TYPE ExampleDomain_Io_In :
STRUCT
END_STRUCT
END_TYPE

(* stored: Version 1.1.0.1
   DUT ExampleDomain_Io_In: Id {ba079b10-98a9-416c-b8c4-6503288d8cd5} *)
